FUNCTION_BLOCK TWO_POS_CONVEYOR_TRANSPORT (* Extracted Composite Function Block Type *)
  (* Standard: 61499-2 *)
  (* Version 4/30/2023, Dmitrii *)
  PACKAGE UAO.Hackathon;
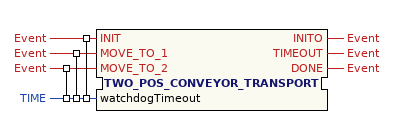
  EVENT_INPUT
    INIT WITH watchdogTimeout; (* Initializes the symbolic link data destination FB with N (1 <= N <= 16) variables *)
    MOVE_TO_1 WITH watchdogTimeout; (* Set Event *)
    MOVE_TO_2 WITH watchdogTimeout; (* Set Event *)
  END_EVENT
  EVENT_OUTPUT
    INITO; (* Initialization confirm *)
    TIMEOUT; (* Delayed Event *)
    DONE; (* Event Output *)
  END_EVENT
  VAR_INPUT
    watchdogTimeout : TIME; (* Delay Time *)
  END_VAR
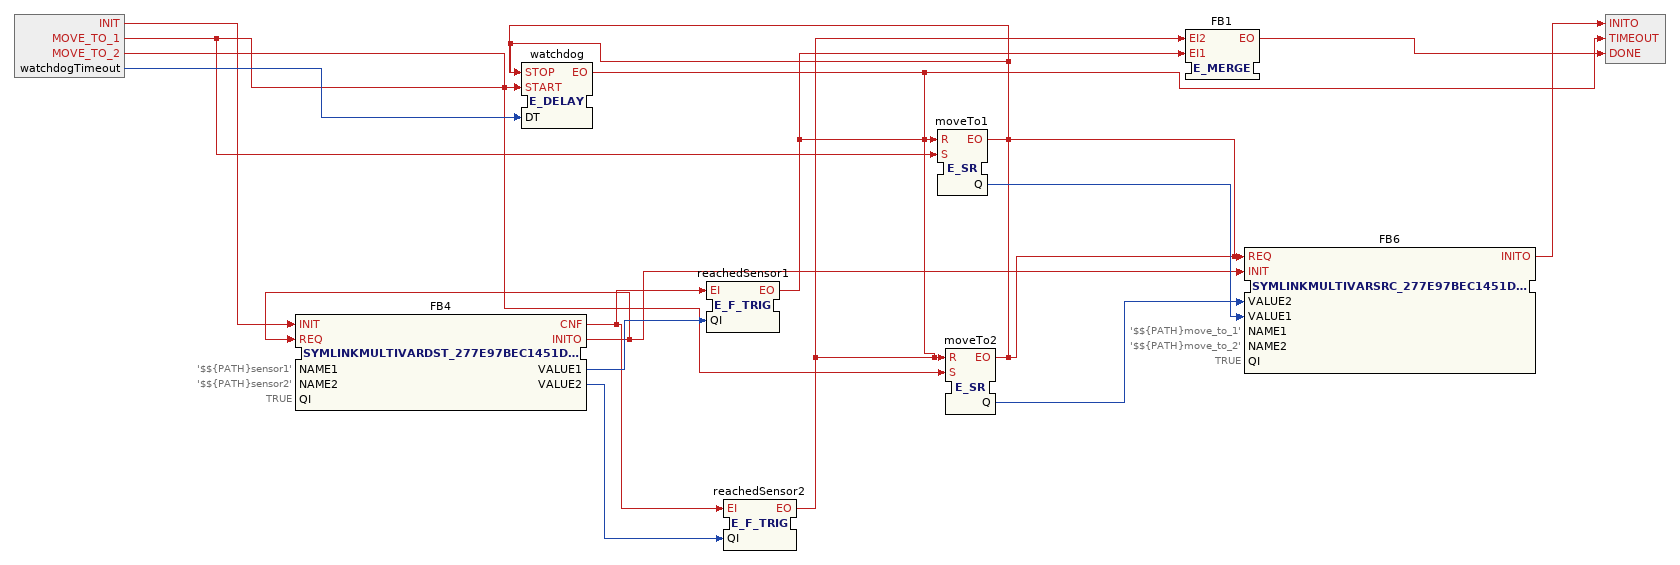
  FBS
    FB4 : SYMLINKMULTIVARDST_277E97BEC1451D2C(NAME1 := '$${PATH}sensor1', NAME2 := '$${PATH}sensor2', QI := TRUE); {SET_ATTRIBUTE(Configuration.GenericFBType.InterfaceParams, Runtime.System#I:=2;VALUE${I$}:BOOL,BOOL)}
    FB6 : SYMLINKMULTIVARSRC_277E97BEC1451D2C(NAME1 := '$${PATH}move_to_1', NAME2 := '$${PATH}move_to_2', QI := TRUE); {SET_ATTRIBUTE(Configuration.GenericFBType.InterfaceParams, Runtime.System#I:=2;VALUE${I$}:BOOL,BOOL)}
    moveTo1 : E_SR;
    moveTo2 : E_SR;
    watchdog : E_DELAY;
    reachedSensor1 : E_F_TRIG;
    reachedSensor2 : E_F_TRIG;
    FB1 : E_MERGE;
  END_FBS
  EVENT_CONNECTIONS
    FB4.CNF TO reachedSensor1.EI;
    FB4.CNF TO reachedSensor2.EI;
    reachedSensor1.EO TO moveTo1.R;
    reachedSensor2.EO TO moveTo2.R;
    moveTo2.EO TO FB6.REQ;
    moveTo1.EO TO FB6.REQ;
    FB4.INITO TO FB6.INIT;
    watchdog.EO TO moveTo1.R;
    watchdog.EO TO moveTo2.R;
    moveTo1.EO TO watchdog.STOP;
    moveTo2.EO TO watchdog.STOP;
    MOVE_TO_1 TO moveTo1.S;
    MOVE_TO_2 TO moveTo2.S;
    watchdog.EO TO TIMEOUT;
    INIT TO FB4.INIT;
    FB6.INITO TO INITO;
    MOVE_TO_1 TO watchdog.START;
    MOVE_TO_2 TO watchdog.START;
    FB4.INITO TO FB4.REQ;
    reachedSensor2.EO TO FB1.EI2;
    FB1.EO TO DONE;
    reachedSensor1.EO TO FB1.EI1;
  END_CONNECTIONS
  DATA_CONNECTIONS
    FB4.VALUE1 TO reachedSensor1.QI;
    FB4.VALUE2 TO reachedSensor2.QI;
    moveTo2.Q TO FB6.VALUE2;
    moveTo1.Q TO FB6.VALUE1;
    watchdogTimeout TO watchdog.DT;
  END_CONNECTIONS
END_FUNCTION_BLOCK
